TYPE ST_IOOutputSimul :
STRUCT
	QxLampeRouge AT%Q*:BOOL;
END_STRUCT
END_TYPE

(* stored: Version 1.1.0.1, ProductVersion 3.1.4020.6
   DUT ST_IOOutputSimul: Id {08e8cc39-f36c-4116-bfb5-3d669fdca8b1} *)
